PROGRAM P4_04_Delete
VAR
	fbPLCDBCmd    	:FB_PLCDBCmdEvt(sNetID:=CONST.AMS_NETID, tTimeout:=DEFAULT_ADS_TIMEOUT);
	sCmdDelete		:STRING[80];
	
	arrParam		:ARRAY [0..5] OF ST_ExpParameter := [(sParaName := 'DateTime', nParaSize := 4, eParaType := E_EXPPARAMETERTYPE.DateTime), 
														(sParaName := 'User', nParaSize := 101, eParaType := E_EXPPARAMETERTYPE.STRING_), 
														(sParaName := 'Event', nParaSize := 101, eParaType := E_EXPPARAMETERTYPE.STRING_), 
														(sParaName := 'Description', nParaSize := 101, eParaType := E_EXPPARAMETERTYPE.STRING_), 
														(sParaName := 'OldValue', nParaSize := 101, eParaType := E_EXPPARAMETERTYPE.STRING_), 
														(sParaName := 'NewValue', nParaSize := 101, eParaType := E_EXPPARAMETERTYPE.STRING_)];
	
	stDBParam 		:ST_AuditTrail;	
END_VAR

sCmdDelete:='DELETE FROM `audit_trail`';
ACT_Cmd();

ACTION ACT_Cmd:
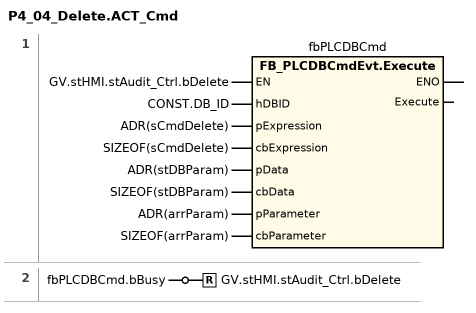
// NETWORK 1
IF GV.stHMI.stAudit_Ctrl.bDelete THEN
    fbPLCDBCmd.Execute(
        hDBID := CONST.DB_ID,
        pExpression := ADR(sCmdDelete),
        cbExpression := SIZEOF(sCmdDelete),
        pData := ADR(stDBParam),
        cbData := SIZEOF(stDBParam),
        pParameter := ADR(arrParam),
        cbParameter := SIZEOF(arrParam));
END_IF

// NETWORK 2
GV.stHMI.stAudit_Ctrl.bDelete R= NOT fbPLCDBCmd.bBusy;
END_ACTION

END_PROGRAM

(* stored: Version 1.1.0.1
   POU P4_04_Delete: Id {af1c0cad-085d-4fc6-8fe7-18299aa6786c}, SpecialFunc None
   Action ACT_Cmd: Id {ed6c2a52-47ad-4667-996f-28147fa826e7} *)
